TYPE ST_Powerstack_MaintenanceParams :
STRUCT
	ForceNetcontactor		: BOOL;
END_STRUCT
END_TYPE

(* stored: Version 1.1.0.1, ProductVersion 3.1.4026.18
   DUT ST_Powerstack_MaintenanceParams: Id {4bdc55f7-f0aa-458a-964b-ed33f950df85} *)
